TYPE
    ComRobIn :
    STRUCT
        {attribute addProperty Name "<#Station bereit fuer Spacer#>"}
        StationClearForSpacer : BOOL;
        {attribute addProperty Name "<#Home Pos erreicht#>"}
        HomePosReached : BOOL;
        {attribute addProperty Name "<#Fehler ID#>"}
        FaultID : INT;
        {attribute addProperty Name "<#Status Running#>"}
        StatusRunning : BOOL;
        {attribute addProperty Name "<#Fehler#>"}
        Fault : BOOL;
        {attribute addProperty Name "<#HighPower aktiv#>"}
        PowerOn : BOOL;
        {attribute addProperty Name "<#EStop aktiv#>"}
        Estop : BOOL;
        {attribute addProperty Name "<#Increase Index#"}
        IncreaseIndex : BOOL;
        {attribute addProperty Name "<#Index Palette Schaumstoffring#>"}
        PalletIndexPick : INT;
        {attribute addProperty Name "<#Berechneter Wert aus Roboter#>"}
        RowPallet : INT;
        {attribute addProperty Name "<#Foto machen#>"}
        TakeFoto : BOOL;
        {attribute addProperty Name "<#Pick Palette Index X#>"}
        PickPalletXcount : INT;
        {attribute addProperty Name "<#Pick Palette Index Y#>"}
        PickPalletYcount : INT;
    END_STRUCT
END_TYPE

(* stored: Version 1.1.0.1, ProductVersion 3.1.4024.12
   DUT ComRobIn: Id {e3ddf2c1-df9f-0e60-14b1-1487ccd4cb19} *)
